FUNCTION F_GenerateData : STRING(255)
VAR_INPUT
END_VAR
VAR
	  fTemperature	: REAL;
	  fHumidity		: REAL;
	  fWindSpeed	: REAL;
	  fbRandom		: DRAND;
	  fbJson 		: FB_JsonSaxWriter;
END_VAR

(* Create random data *)
fbRandom(Seed := 1, Num => fTemperature);
fbRandom(Seed := 2, Num => fHumidity);
fbRandom(Seed := 3, Num => fWindSpeed);
fTemperature := fTemperature * 100;
fHumidity := fHumidity * 10;
fWindSpeed := fWindSpeed + 20.42;

(* Create JSON document and embed generated data *)
fbJson.StartObject();
fbJson.AddKey('DeviceId');
fbJson.AddString(GVL.sDeviceId);
fbJson.AddKey('Temperature');
fbJson.AddReal(fTemperature);
fbJson.AddKey('Humidity');
fbJson.AddReal(fHumidity);
fbJson.AddKey('WindSpeed');
fbJson.AddReal(fWindSpeed);
fbJson.EndObject();
F_GenerateData := fbJson.GetDocument();

END_FUNCTION

(* stored: Version 1.1.0.1, ProductVersion 3.1.4022.3
   POU F_GenerateData: Id {7e0d66fa-b0f0-4666-b14c-fa381f027f98}, SpecialFunc None *)
